{attribute addProperty BoxType "EK1122-0000-0018"}
{attribute addProperty Id "Beckhoff_EL66xxsub_EK1100EK1100_179A0949162A_0032_EL6690_0002_0000EL6690_DEF6788A263.25A_0033_EL6690_0002_0016EL6690_DEF6788A263.25A_0034_EL6690_0002_0017EL6690_DEF6788A263.25A_0035_EL6690_0002_0018EL6690_DEF6788A263.25A_0036_EL6690_0002_0019EL6690_DEF6788A263.25A_0040_EL6692_0002_0016EL6692_4FA89B0317822.25A_0041_EL6692_0002_0017EL6692_4FA89B0317822.25A_0042_EL6692_0002_0018EL6692_4FA89B0317822.25A_0043_EL6692_0002_0019EL6692_4FA89B0317822.25A_0044_EL6692_0002_0020EL6692_67810D9517822.25A_0046_EL6695_0002_0001EL6695_5B9A4EC315419.25A_0048_EL6695_0002_0002EL6695_5B9A4EC315419.25A_0050_EL6695_0002_0003EL6695_5B9A4EC315419.25A_0052_EL6695_0002_0004EL6695_5B9A4EC315419.25A_0054_EL6695_0002_0005EL6695_5B9A4EC315419.25A_0056_EL6695_0002_0006EL6695_5B9A4EC315419.25"}
{attribute addProperty CRC "3594126091"}
{attribute addProperty SizeInBites "1960"}
{attribute addProperty SizeInBytes "245"}
TYPE Beckhoff_EL66xxEK1122_D63A030B EXTENDS EK1122_179A0949 :
STRUCT
	{attribute addProperty Name "Beckhoff_EL66xxsub_EK1100"}
	Beckhoff_EL66xxsub_EK1100 : EK1100_179A0949;
	{attribute addProperty Name "A_0032_EL6690_0002_0000"}
	A_0032_EL6690_0002_0000 : EL6690_DEF6788A;
	{attribute addProperty Name "A_0033_EL6690_0002_0016"}
	A_0033_EL6690_0002_0016 : EL6690_DEF6788A;
	{attribute addProperty Name "A_0034_EL6690_0002_0017"}
	A_0034_EL6690_0002_0017 : EL6690_DEF6788A;
	{attribute addProperty Name "A_0035_EL6690_0002_0018"}
	A_0035_EL6690_0002_0018 : EL6690_DEF6788A;
	{attribute addProperty Name "A_0036_EL6690_0002_0019"}
	A_0036_EL6690_0002_0019 : EL6690_DEF6788A;
	{attribute addProperty Name "A_0040_EL6692_0002_0016"}
	A_0040_EL6692_0002_0016 : EL6692_4FA89B03;
	{attribute addProperty Name "A_0041_EL6692_0002_0017"}
	A_0041_EL6692_0002_0017 : EL6692_4FA89B03;
	{attribute addProperty Name "A_0042_EL6692_0002_0018"}
	A_0042_EL6692_0002_0018 : EL6692_4FA89B03;
	{attribute addProperty Name "A_0043_EL6692_0002_0019"}
	A_0043_EL6692_0002_0019 : EL6692_4FA89B03;
	{attribute addProperty Name "A_0044_EL6692_0002_0020"}
	A_0044_EL6692_0002_0020 : EL6692_67810D95;
	{attribute addProperty Name "A_0046_EL6695_0002_0001"}
	A_0046_EL6695_0002_0001 : EL6695_5B9A4EC3;
	{attribute addProperty Name "A_0048_EL6695_0002_0002"}
	A_0048_EL6695_0002_0002 : EL6695_5B9A4EC3;
	{attribute addProperty Name "A_0050_EL6695_0002_0003"}
	A_0050_EL6695_0002_0003 : EL6695_5B9A4EC3;
	{attribute addProperty Name "A_0052_EL6695_0002_0004"}
	A_0052_EL6695_0002_0004 : EL6695_5B9A4EC3;
	{attribute addProperty Name "A_0054_EL6695_0002_0005"}
	A_0054_EL6695_0002_0005 : EL6695_5B9A4EC3;
	{attribute addProperty Name "A_0056_EL6695_0002_0006"}
	A_0056_EL6695_0002_0006 : EL6695_5B9A4EC3;
END_STRUCT
END_TYPE

(* stored: Version 1.2.0.0, ProductVersion 3.1.4024.9
   DUT Beckhoff_EL66xxEK1122_D63A030B: Id {2e5b303b-cd33-4f87-8e8c-12c3e6a35aa8} *)
